// TIA Portal V17 export
// export: Created 2025-01-08T13:55:36.8986241Z, ExportSetting WithDefaults, DisplayName Totally Integrated Automation Portal, DisplayVersion V17, DisplayName TIA Portal Openness, DisplayVersion V17, DisplayName TIA Portal Version Control Interface, DisplayVersion V17, DisplayName SINAMICS Startdrive Advanced, DisplayVersion V17 Update2, DisplayName SINAMICS Startdrive G130, G150, S120, S150, SINAMICS MV, S210, DisplayVersion V17 Update2, DisplayName SINAMICS Startdrive G110M, G120, G120C, G120D, G120P, G115D, DisplayVersion V17 Update2, DisplayName STEP 7 Professional, DisplayVersion V17, DisplayName STEP 7 Safety, DisplayVersion V17, DisplayName WinCC Advanced, DisplayVersion V17
TYPE "HSMMachineParaMask2"
// stored: IsFailsafeCompliant false
   STRUCT
      iExternalStart : Bool;
      iLowLabelInput : Bool;
      iRibbonInput : Bool;
      iSyncParameter : Bool;
      iSyncOutputDelay : Bool;
      iSyncOutputLenght : Bool;
      iZeroDownTimeMode : Bool;
      iZeroDownTimeSensorDistance : Bool;
      iRestLenghtOnLowLabel : Bool;
      iLowLabelSensorPolarity : Bool;
      iWebBreakSensorPolarity : Bool;
      iWarningOutputPolarity : Bool;
      iSync2Parameter : Bool;
      iSync2OutputDelay : Bool;
      iSync2OutputLenght : Bool;
      iSync3Parameter : Bool;
   END_STRUCT;
END_TYPE
